{attribute 'GeneratedUsingTerminal: EP9128-0021-0018'}
{attribute addProperty BoxType "EP9128-0021-0018"}
{attribute addProperty Id "A_0013_EP9128_0021_0019A_0013_EP9128_0021_0019_9F59C97D579A_0010_EP9128_0021_0018_2_EP9128_1021EP9128_AB5A94672A_0010_EP9128_0021_0018_3_EP9128_2021EP9128_AB5A94672"}
{attribute addProperty CRC "2910415530"}
{attribute addProperty Size "583"}
TYPE A_0010_EP9128_0021_0018_AD796AAA EXTENDS EP9128_AB5A9467 :
STRUCT
	{attribute addProperty Name "A_0013_EP9128_0021_0019"}
	A_0013_EP9128_0021_0019 : A_0013_EP9128_0021_0019_9F59C97D;
	{attribute addProperty Name "A_0010_EP9128_0021_0018_2_EP9128_1021"}
	A_0010_EP9128_0021_0018_2_EP9128_1021 : EP9128_AB5A9467;
	{attribute addProperty Name "A_0010_EP9128_0021_0018_3_EP9128_2021"}
	A_0010_EP9128_0021_0018_3_EP9128_2021 : EP9128_AB5A9467;
END_STRUCT
END_TYPE

(* stored: Version 1.2.0.0, ProductVersion 3.1.4024.9
   DUT A_0010_EP9128_0021_0018_AD796AAA: Id {a62325a3-b2eb-4588-9e57-ce70d2750765} *)
